{attribute 'GeneratedUsingTerminal: EP6601-0002-0018'}
{attribute addProperty BoxType "EP6601-0002-0018"}
{attribute addProperty Id "InfoDataAT %I*InfoData_32EB74EA10"}
{attribute addProperty CRC "4004708084"}
{attribute addProperty Size "10"}
TYPE EP6601_EEB2FEF4 EXTENDS EtcSlaveTerminalBase_947E5A46 :
STRUCT
	{attribute addProperty Name "InfoData"}
	InfoData : InfoData_32EB74EA;
END_STRUCT
END_TYPE

(* stored: Version 1.2.0.0, ProductVersion 3.1.4024.9
   DUT EP6601_EEB2FEF4: Id {55199e7f-edaf-469a-a7c0-074fc786fdc3} *)
